	comm.Publish('telescope', 'dome', 'Mirror1Temperature',	LREAL_TO_FMTSTR(temperature_mirror1, 2, TRUE));
	comm.Publish('telescope', 'dome', 'Mirror2Temperature',	LREAL_TO_FMTSTR(temperature_mirror2, 2, TRUE));
	
	MQTTTimer(IN:=FALSE);

END_IF

END_PROGRAM

// ---- GlobalTextList.TcGTLO
TEXTLIST GlobalTextList
  265 = '%.0f %'
  500 = '%.0f%'
  194 = '%.2f'
  730 = '%.2f mm'
  1120 = '%.2f °'
  943 = '%.2f °/s'
  1152 = '%.2f°'
  465 = '%.2f°/s'
  234 = '%.4'
  1272 = '%.4 °'
  484 = '%.4f'
  144 = '%.4f '
  339 = '%.4f mm'
  848 = '%.4f °'
  941 = '%.4f°'
  616 = '%d'
  792 = '%s'
  78 = '+'
  114 = '-'
  170 = '/'
  643 = '22'
  411 = 'Alt'
  207 = 'Altitude'
  148 = 'Automatic'
  1021 = 'Azimuth'
  785 = 'Azimuth:'
  247 = 'Brake'
  911 = 'Brake clearing'
  798 = 'Brake closed'
  396 = 'Brake open'
  958 = 'Brakes'
  272 = 'busy'
  573 = 'Busy'
  619 = 'Calculated'
  688 = 'Calibrated'
  337 = 'Close'
  41 = 'Close brake'
  507 = 'Closed'
  361 = 'Closing'
  392 = 'Cold'
  12 = 'Cover 1'
  678 = 'Cover 2'
  857 = 'Cover 3'
  816 = 'Current'
  1081 = 'Declination'
  815 = 'Derotator:'
  524 = 'Diag: %s'
  957 = 'Direction error'
  511 = 'Drive   Error'
  101 = 'EL1904'
  761 = 'EL2904'
  409 = 'Elevation:'
  894 = 'Enable'
  686 = 'EnabParkle'
  562 = 'Equatorial'
  868 = 'ErrAck'
  879 = 'Error'
  225 = 'Estop: %s'
  755 = 'Far'
  479 = 'Global'
  548 = 'GoHome'
  867 = 'GoTo'
  331 = 'High'
  940 = 'Homed'
  483 = 'Homing'
  1063 = 'Horizontal'
  81 = 'Hot'
  163 = 'Level'
  846 = 'Level:'
  557 = 'Limits'
  58 = 'Low'
  697 = 'Manual'
  389 = 'Motor #1'
  611 = 'Motor #2'
  712 = 'Move'
  466 = 'Movement'
  765 = 'Moving'
  59 = 'Near'
  33 = 'Oil cold'
  995 = 'Oil high'
  856 = 'Oil hot'
  768 = 'Oil low'
  37 = 'Oil pan maximum'
  481 = 'Oil pressure OK'
  874 = 'Oil Status'
  498 = 'Oil warning'
  366 = 'Open'
  482 = 'Open brake'
  1197 = 'Open/Close'
  186 = 'Opening'
  352 = 'Override Start Pump'
  744 = 'Override Start Sucction'
  606 = 'Override stop pump'
  890 = 'Overrides'
  384 = 'Pan max'
  273 = 'park'
  92 = 'Park'
  1353 = 'Parked'
  525 = 'Position'
  919 = 'Power'
  641 = 'Pressure'
  196 = 'Pump'
  523 = 'Pump running'
  120 = 'ready'
  176 = 'Ready'
  685 = 'Reset'
  789 = 'Restart'
  1221 = 'Right Ascension'
  360 = 'Roof'
  456 = 'Roof #1'
  944 = 'Roof #2'
  104 = 'Safety Diag%s'
  521 = 'Safety Diag: %s'
  672 = 'Safety State: %s'
  309 = 'Set'
  777 = 'slew'
  1245 = 'Slew'
  724 = 'Slewing'
  717 = 'sliding'
  138 = 'Slow close'
  996 = 'Slow open'
  49 = 'Speed'
  566 = 'Start'
  202 = 'Start Sucction'
  520 = 'State'
  809 = 'State: %s'
  354 = 'Status'
  328 = 'STO ErrAck:'
  540 = 'STO Reset:'
  488 = 'STO:'
  572 = 'Stop'
  189 = 'Stop pump'
  155 = 'stopped'
  790 = 'Stopped'
  614 = 'Sucction'
  782 = 'Sucction running'
  704 = 'Succtionrunning'
  385 = 'Sync error'
  362 = 'track'
  569 = 'Track'
  364 = 'tracking'
  356 = 'Tracking'
  136 = 'Unlocked'
  67 = 'Velocity'
  480 = 'Warning'
  609 = 'Zero counter'
  1015 = ']'
END_TEXTLIST

// ---- VISUs/Hydraulics.TcVIS
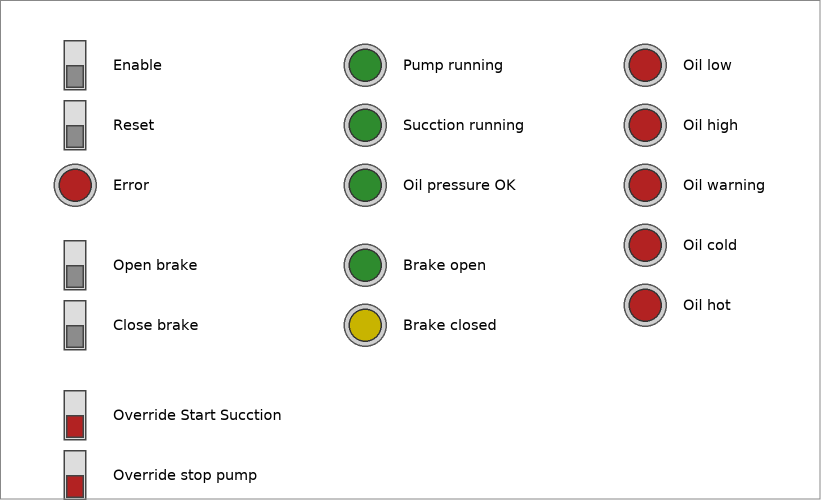
VISUALIZATION Hydraulics  // 821x500
    DipSwitch (50,40 50x50), variable: HydraulicsControl.enable, behaviour: TOGGLE, style: Switch-DipSwitch-Gray
    DipSwitch (50,100 50x50), variable: HydraulicsControl.reset, behaviour: TOGGLE, style: Switch-DipSwitch-Gray
    Label (110,50 101x30), "Enable"
    Label (110,110 101x30), "Reset"
    Lamp1 (50,160 50x50), variable: HydraulicsControl.error, style: Lamp-Lamp1-Red
    Label (110,170 101x30), "Error"
    DipSwitch (50,390 50x50), variable: HydraulicsControl.suction_manual, behaviour: TOGGLE, style: Switch-DipSwitch-Red
    DipSwitch (50,450 50x50), variable: HydraulicsControl.pump_manual_stop, behaviour: TOGGLE, style: Switch-DipSwitch-Red
    Label (110,400 171x30), "Override Start Sucction"
    Label (110,460 161x30), "Override stop pump"
    Lamp1 (340,40 50x50), variable: HydraulicsControl.pump_running, style: Lamp-Lamp1-Green
    Label (400,50 141x30), "Pump running"
    Lamp1 (340,100 50x50), variable: HydraulicsControl.suction_running, style: Lamp-Lamp1-Green
    Label (400,110 141x30), "Sucction running"
    Lamp1 (340,240 50x50), variable: HydraulicsControl.brake_open, style: Lamp-Lamp1-Green
    Label (400,250 141x30), "Brake open"
    Lamp1 (340,300 50x50), variable: HydraulicsControl.brake_closed, style: Lamp-Lamp1-Yellow
    Label (400,310 141x30), "Brake closed"
    Lamp1 (620,40 50x50), variable: HydraulicsControl.oil_low, style: Lamp-Lamp1-Red
    Label (680,50 141x30), "Oil low"
    Lamp1 (620,100 50x50), variable: HydraulicsControl.oil_high, style: Lamp-Lamp1-Red
    Label (680,110 141x30), "Oil high"
    Lamp1 (620,160 50x50), variable: HydraulicsControl.oil_warning, style: Lamp-Lamp1-Red
    Label (680,170 141x30), "Oil warning"
    Lamp1 (340,160 50x50), variable: HydraulicsControl.oil_pressure_OK, style: Lamp-Lamp1-Green
    Label (400,170 141x30), "Oil pressure OK"
    Lamp1 (620,220 50x50), variable: HydraulicsControl.oil_cold, style: Lamp-Lamp1-Red
    Label (680,230 141x30), "Oil cold"
    Lamp1 (620,280 50x50), variable: HydraulicsControl.oil_hot, style: Lamp-Lamp1-Red
    Label (680,290 141x30), "Oil hot"
    DipSwitch (50,240 50x50), variable: HydraulicsControl.iopen_brake, behaviour: TOGGLE, style: Switch-DipSwitch-Gray
    DipSwitch (50,300 50x50), variable: HydraulicsControl.iclose_brake, behaviour: TOGGLE, style: Switch-DipSwitch-Gray
    Label (110,250 101x30), "Open brake"
    Label (110,310 101x30), "Close brake"
END_VISUALIZATION

// ---- VISUs/Safety.TcVIS
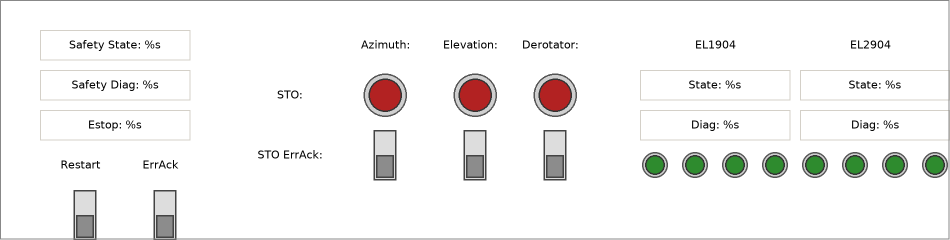
VISUALIZATION Safety  // 950x240
    Label (340,30 91x30), "Azimuth:"
    Lamp1 (360,70 50x50), variable: MAIN.AzimuthControl.IbSTO, style: Lamp-Lamp1-Red
    Label (430,30 81x30), "Elevation:"
    Lamp1 (450,70 50x50), variable: MAIN.ElevationControl.IbSTO, style: Lamp-Lamp1-Red
    Label (510,30 81x30), "Derotator:"
    Lamp1 (530,70 50x50), variable: MAIN.DerotatorControl.IbSTO, style: Lamp-Lamp1-Red
    Label (240,80 100x30), "STO:"
    DipSwitch (60,190 50x50), variable: MAIN.SafetyHandling.outRestart, behaviour: TOGGLE, style: Switch-DipSwitch-Gray
    DipSwitch (530,130 50x50), variable: MAIN.SafetyHandling.outResetDerotatorSTO, behaviour: TOGGLE, style: Switch-DipSwitch-Gray
    DipSwitch (360,130 50x50), variable: MAIN.SafetyHandling.outResetAzimuthSTO, behaviour: TOGGLE, style: Switch-DipSwitch-Gray
    DipSwitch (450,130 50x50), variable: MAIN.SafetyHandling.outResetElevationSTO, behaviour: TOGGLE, style: Switch-DipSwitch-Gray
    Label (240,140 100x30), "STO ErrAck:"
    Label (40,150 81x30), "Restart"
    DipSwitch (140,190 50x50), variable: MAIN.SafetyHandling.outErrAck, behaviour: TOGGLE, style: Switch-DipSwitch-Gray
    Label (120,150 81x30), "ErrAck"
    Textfield (40,30 150x30), "Safety State: %s", text variable: MAIN.SafetyHandling.fbInfoEStop1.sState, input disabled if: TRUE
    Textfield (40,110 150x30), "Estop: %s", text variable: MAIN.SafetyHandling.fbInfoEStop1.sState, input disabled if: TRUE
    Textfield (40,70 150x30), "Safety Diag: %s", text variable: MAIN.SafetyHandling.fbInfoEStop1.sDiag, input disabled if: TRUE
    Label (670,30 91x30), "EL1904"
    Label (830,30 81x30), "EL2904"
    Textfield (640,70 150x30), "State: %s", text variable: MAIN.SafetyHandling.fbInfoSafetyIn.sState, input disabled if: TRUE
    Textfield (640,110 150x30), "Diag: %s", text variable: MAIN.SafetyHandling.fbInfoSafetyIn.sDiag, input disabled if: TRUE
    Textfield (800,70 150x30), "State: %s", text variable: MAIN.SafetyHandling.fbInfoSafetyOut.sState, input disabled if: TRUE
    Textfield (800,110 150x30), "Diag: %s", text variable: MAIN.SafetyHandling.fbInfoSafetyOut.sDiag, input disabled if: TRUE
    Lamp1 (640,150 30x30), variable: MAIN.SafetyHandling.bSafetyInCh1, style: Lamp-Lamp1-Green
    Lamp1 (680,150 30x30), variable: MAIN.SafetyHandling.bSafetyInCh2, style: Lamp-Lamp1-Green
    Lamp1 (720,150 30x30), variable: MAIN.SafetyHandling.bSafetyInCh3, style: Lamp-Lamp1-Green
    Lamp1 (760,150 30x30), variable: MAIN.SafetyHandling.bSafetyInCh4, style: Lamp-Lamp1-Green
    Lamp1 (800,150 30x30), variable: MAIN.SafetyHandling.bSafetyInCh1, style: Lamp-Lamp1-Green
    Lamp1 (840,150 30x30), variable: MAIN.SafetyHandling.bSafetyInCh2, style: Lamp-Lamp1-Green
    Lamp1 (880,150 30x30), variable: MAIN.SafetyHandling.bSafetyInCh3, style: Lamp-Lamp1-Green
    Lamp1 (920,150 30x30), variable: MAIN.SafetyHandling.bSafetyInCh4, style: Lamp-Lamp1-Green
END_VISUALIZATION

// ---- VISUs/Visualization.TcVIS
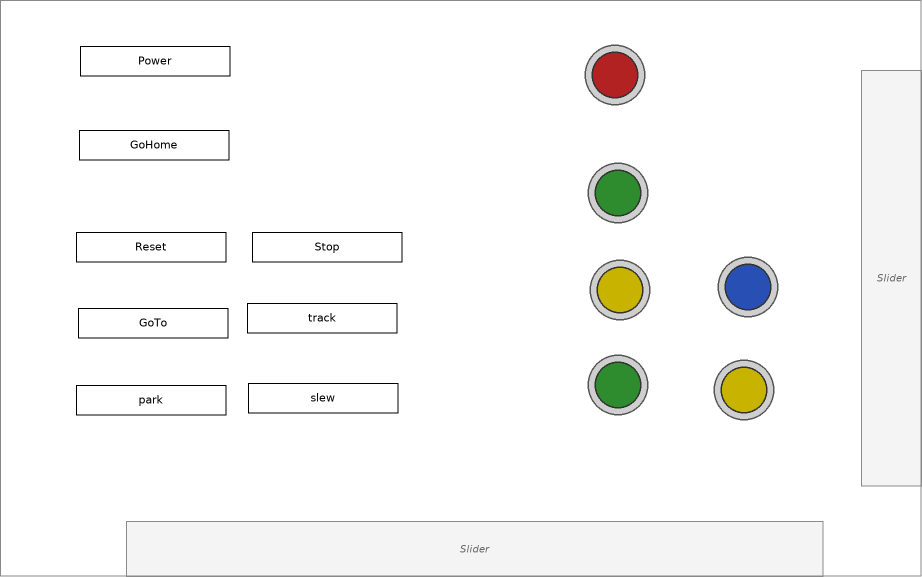
VISUALIZATION Visualization  // 922x577
    RoundedRectangle (80,46 150x30), "Power", colour toggle: TelescopeControl.power
        toggle TelescopeControl.power
    Rectangle (79,130 150x30), "GoHome", colour toggle: TelescopeControl.gohome
        toggle TelescopeControl.gohome
    Lamp1 (580,40 70x70), tooltip "Error", variable: TelescopeControl.error, style: Lamp-Lamp1-Red
    Lamp1 (583,158 70x70), tooltip "ready", variable: TelescopeControl.ready, style: Lamp-Lamp1-Green
    Rectangle (76,232 150x30), "Reset", colour toggle: TelescopeControl.reset
        toggle TelescopeControl.reset
    RoundedRectangle (78,308 150x30), "GoTo", colour toggle: TelescopeControl.goto
        toggle TelescopeControl.goto
    Lamp1 (585,255 70x70), tooltip "sliding", variable: TelescopeControl.sliding, style: Lamp-Lamp1-Yellow
    RoundedRectangle (76,385 150x30), "park", colour toggle: TelescopeControl.park
        toggle TelescopeControl.park
    Lamp1 (583,350 70x70), tooltip "stopped", variable: TelescopeControl.Safetypped, style: Lamp-Lamp1-Green
    Slider (126,521 697x56), variable: TelescopeControl.rightascension, scale 0..360
    Slider (861,70 61x416), variable: TelescopeControl.declination, scale -90..90
    Lamp1 (713,252 70x70), tooltip "tracking", variable: TelescopeControl.tracking, style: Lamp-Lamp1-Blue
    RoundedRectangle (247,303 150x30), "track", colour toggle: TelescopeControl.track
        toggle TelescopeControl.track
    RoundedRectangle (248,383 150x30), "slew", colour toggle: TelescopeControl.slew
        toggle TelescopeControl.slew
    Lamp1 (709,355 70x70), tooltip "busy", variable: TelescopeControl.busy, style: Lamp-Lamp1-Yellow
    RoundedRectangle (252,232 150x30), "Stop", colour toggle: TelescopeControl.Safetyp
        toggle TelescopeControl.stop
END_VISUALIZATION
